Fanuc KAREL source: kt00295.KL

-- PROVISIONAL review KL for V1013-1; original PC SHA256 3ed75ae5501f83f2ce387c24fc29bf74c9c0e140b9f0148ad240bf643505a002
-- Incomplete behavior may be omitted. Consult companion uncertainty JSON. Do not deploy.
PROGRAM KT00295
%NOLOCKGROUP
VAR
  I1 : INTEGER
  OUT : BOOLEAN
-- UNRESOLVED_DECL Y2 type=002018
BEGIN
  -- UNRESOLVED_PC offsets 5-16; opcodes 2E,23
  -- UNRESOLVED_PC offsets 21-35; opcodes 2E,22,9D,33,B2
  -- UNRESOLVED_PC offsets 40-62; opcodes 21,22,9D,33,B1,58,23
  -- UNRESOLVED_PC offsets 67-71; opcodes 7F
END KT00295
